// TwinCAT 3 PLC project DialogPLC
// ProgramVersion: 3.1.4022.4
// libraries:
//   Tc2_Standard, * (Beckhoff Automation GmbH)
//   Tc2_System, * (Beckhoff Automation GmbH)
//   Tc3_Module, * (Beckhoff Automation GmbH)
//   VisuDialogs, * (System)
//   VisuSymbols,3.5.10.0,System
// project tree:
//   / GlobalTextList.TcGTLO, PlcTask.TcTTO, Visualization Manager.TcVMO (not stored), VISU_TASK.TcTTO
//   GVLs/ GVL.TcGVL
//   POUs/ CloseMessageDialog.TcPOU, MAIN.TcPOU, OpenMessageDialog.TcPOU, P_Dialog.TcPOU
//   VISUs/ DialogTest.TcVIS, Visualization2.TcVIS
// real-time tasks:
//   TASK PlcTask: cycle T#10ms, priority 20, ADS port 350
//   TASK VISU_TASK: cycle T#200000us, priority 30, ADS port 351

CONFIGURATION DialogPLC
    RESOURCE PLC ON TwinCAT3
        TASK PlcTask(INTERVAL := T#10ms, PRIORITY := 20);
        TASK VISU_TASK(INTERVAL := T#200000us, PRIORITY := 30);
        PROGRAM MAIN WITH PlcTask : MAIN;
        PROGRAM VisuElems_Visu_Prg WITH VISU_TASK : VisuElems.Visu_Prg;
    END_RESOURCE
END_CONFIGURATION

// ---- GVLs/GVL.TcGVL
{attribute 'qualified_only'}
VAR_GLOBAL
	sTitle : STRING := 'Message ...';
	result : VisuElems.Visu_DialogResult;
	iDialogManager : VisuElems.IDialogManager;
	iMessageDialog : VisuElems.IVisualisationDialog;
END_VAR

// ---- POUs/MAIN.TcPOU
PROGRAM MAIN
VAR
END_VAR

P_Dialog();

END_PROGRAM

// ---- POUs/P_Dialog.TcPOU
PROGRAM P_Dialog
VAR
	nXPos 			: INT:=200; //pozycja popup na ekranie
	nYPos 			: INT:=200; //pozycja popup na ekranie
	fbOpenTrigger 	: R_TRIG;
	bClose 			: BOOL;
	fbCloseTrigger 	: R_TRIG;
	sMessage		: STRING;
	bOpen			: BOOL;
	sResult			: STRING;
	bVisible		: BOOl;
	tof1			: TOF;
	ftResult		: F_TRIG;
	bSwitchParameter: BOOL;
	nCount			: INT;
END_VAR

IF bSwitchParameter THEN
	sMessage:='Parameter text 111111';
ELSE
	sMessage:='Parameter text 222222';
END_IF


fbOpenTrigger(CLK :=bOpen);
IF fbOpenTrigger.Q THEN
	OpenMessageDialog(sMessage := sMessage);
	bOpen:=FALSE;
END_IF

fbCloseTrigger(CLK := bClose);
IF fbCloseTrigger.Q THEN
	nCount := nCount + 1;
	CloseMessageDialog();
	bClose:=FALSE;
END_IF


IF GVL.iMessageDialog <> 0 THEN
	GVL.result := GVL.iMessageDialog.GetResult();
END_IF


IF GVL.result = VisuElemsWinControls.Visu_DialogResult.OK THEN
	sResult:='You clicked OK'; 
END_IF

IF GVL.result = VisuElemsWinControls.Visu_DialogResult.Cancel THEN
	sResult:='You clicked Cancel'; 
END_IF

tof1(IN:=bVisible, PT:=T#1S);

bVisible:=FALSE;

END_PROGRAM

// ---- POUs/OpenMessageDialog.TcPOU
FUNCTION OpenMessageDialog : BOOL
VAR_INPUT
	sMessage: STRING;
END_VAR
VAR
	pMessageInfo : POINTER TO DialogTest_VISU_STRUCT; // "MessageDialog" _VISU_STRUCT contains the parameters defined in the interface of visualization "MessageDialog"
	stMyRect : VisuElems.VisuStructSimpleRectangle;
	pTempClientData : POINTER TO VisuElems.VisuStructClientData;
	pLastClientData : POINTER TO VisuElems.VisuStructClientData;
	nIteratorSave : INT;
	nCounter : INT;
		result : VisuElems.Visu_DialogResult;
END_VAR

nIteratorSave := VisuElems.VisuElemBase.Visu_Globals.g_ClientManager.SaveIteration(); 
VisuElems.VisuElemBase.Visu_Globals.g_ClientManager.BeginIteration();

GVL.iDialogManager := VisuElems.VisuElemBase.g_VisuManager.GetDialogManager();

// Assign the argument in all currently active clients
pTempClientData := VisuElems.VisuElemBase.Visu_Globals.g_ClientManager.GetNextClient();

WHILE pTempClientData <> 0 DO
	GVL.iMessageDialog := GVL.iDialogManager.GetDialog('DialogTest'); // dialog to be handled is specified
	IF GVL.iMessageDialog <> 0 THEN
		GVL.iMessageDialog.SetResult(result);
		pMessageInfo := GVL.iDialogManager.GetClientInterface(GVL.iMessageDialog, pTempClientData);
		IF pMessageInfo <> 0 THEN      // in the following the parameters of the message dialog will be read from the Message_VISU_STRUCT
			pMessageInfo^.sText := sMessage;
		END_IF
	END_IF 
	
	pLastClientData := pTempClientData;
	pTempClientData := VisuElems.VisuElemBase.g_ClientManager.GetNextClient();
	nCounter := nCounter + 1;
END_WHILE

// Open Dialog on all Clients
GVL.iMessageDialog := GVL.iDialogManager.GetDialog('DialogTest'); // dialog to be handled is specified
IF GVL.iMessageDialog <> 0 THEN
	stMyRect.ptTopLeft.iX := P_Dialog.nXPos;
	stMyRect.ptTopLeft.iY := P_Dialog.nYPos;
	stMyRect.ptBottomRight.iX := 10;
	stMyRect.ptBottomRight.iY := 10;
	GVL.iDialogManager.OpenDialog3(GVL.iMessageDialog, pLastClientData, TRUE, ADR(stMyRect), 0, VisuElems.Visu_InputFlags.GlobalOpenCloseDialog);
END_IF

VisuElems.VisuElemBase.Visu_Globals.g_ClientManager.RestoreIteration(nIteratorSave);

END_FUNCTION

// ---- POUs/CloseMessageDialog.TcPOU
FUNCTION CloseMessageDialog : BOOL
VAR_INPUT
	//pClientData : POINTER TO VisuElems.VisuStructClientData;
END_VAR
VAR
	iDialogManager2 : VisuElems.IDialogManager2 := 0;
	pClientData 	: POINTER TO VisuElems.VisuStructClientData;
	nIteratorSave 	: INT;
END_VAR



nIteratorSave := VisuElems.VisuElemBase.Visu_Globals.g_ClientManager.SaveIteration(); 
VisuElems.VisuElemBase.Visu_Globals.g_ClientManager.BeginIteration();
GVL.iDialogManager := VisuElems.VisuElemBase.g_VisuManager.GetDialogManager();
pClientData := VisuElems.VisuElemBase.Visu_Globals.g_ClientManager.GetNextClient();

// Cloase Dialog on all Clients
IF pClientData <> 0 THEN
	GVL.iMessageDialog := GVL.iDialogManager.GetDialog('DialogTest'); // dialog to be handled is specified
	IF GVL.iMessageDialog <> 0 THEN
		IF (iDialogManager2 = 0) THEN
			__QUERYINTERFACE(VisuElems.g_VisuManager.GetDialogManager(), iDialogManager2);
		END_IF
		GVL.result := GVL.iMessageDialog.GetResult();
		IF (iDialogManager2 <> 0) THEN
			iDialogManager2.CloseDialog2(GVL.iMessageDialog, pClientData, VisuElems.Visu_InputFlags.GlobalOpenCloseDialog);
		ELSE
			GVL.iDialogManager.CloseDialog(GVL.iMessageDialog, pClientData);	// Closes The Dialog on all "pClientData"	
		END_IF
	END_IF
END_IF

VisuElems.VisuElemBase.Visu_Globals.g_ClientManager.RestoreIteration(nIteratorSave);

END_FUNCTION

// ---- GlobalTextList.TcGTLO
TEXTLIST GlobalTextList
  242 = '%s'
  244 = 'Cancel'
  137 = 'Close'
  243 = 'OK'
  76 = 'Open'
  255 = 'Open Dialog'
  345 = 'Open Dialog BOX'
  907 = 'Switch parameter'
  801 = 'VIsu1'
  640 = 'VIsu2'
END_TEXTLIST

// ---- VISUs/DialogTest.TcVIS
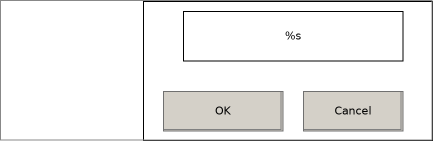
VISUALIZATION DialogTest  // 433x141
VAR_INPUT
	sText: string;
END_VAR
    Rectangle (143,1 290x140)
    Rectangle (183,11 220x50), "%s", text variable: sText
    Button (163,91 120x40), "OK"
        OnDialogClosed: execute { P_Dialog.bVisible:=TRUE; P_Dialog.bClose:=TRUE; }
        OnMouseClick: CloseDialog Dialog=DialogTest, Result=OK, NumpadKeypadSet=True
    Button (303,91 100x40), "Cancel"
        OnDialogClosed: execute { P_Dialog.bVisible:=TRUE; P_Dialog.bClose:=TRUE; }
        OnMouseClick: CloseDialog Dialog=DialogTest, Result=Cancel, NumpadKeypadSet=True
END_VISUALIZATION

// ---- VISUs/Visualization2.TcVIS
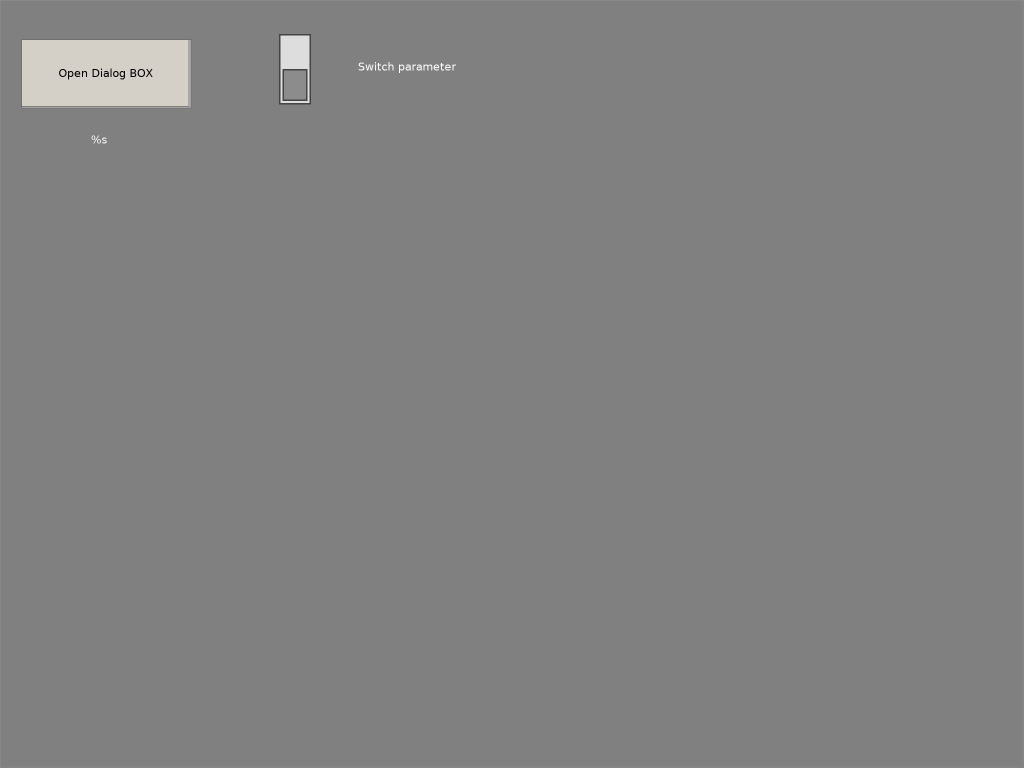
VISUALIZATION Visualization2  // 1024x768
    Button (21,39 170x69), "Open Dialog BOX"
        tap P_Dialog.bOpen
    Rectangle (24,125 150x30), "%s", text variable: P_Dialog.sResult, invisible if: Not P_Dialog.bVisible
    DipSwitch (260,34 70x70), variable: P_Dialog.bSwitchParameter, behaviour: TOGGLE, style: Switch-DipSwitch-Gray
    Label (332,52 150x30), "Switch parameter"
END_VISUALIZATION
